// Mitsubishi GX Works2 project: Unloader Panel 23.07.21   PLC: Q03UDV
// Unloader Panel 23.07.21

PROGRAM MAIN
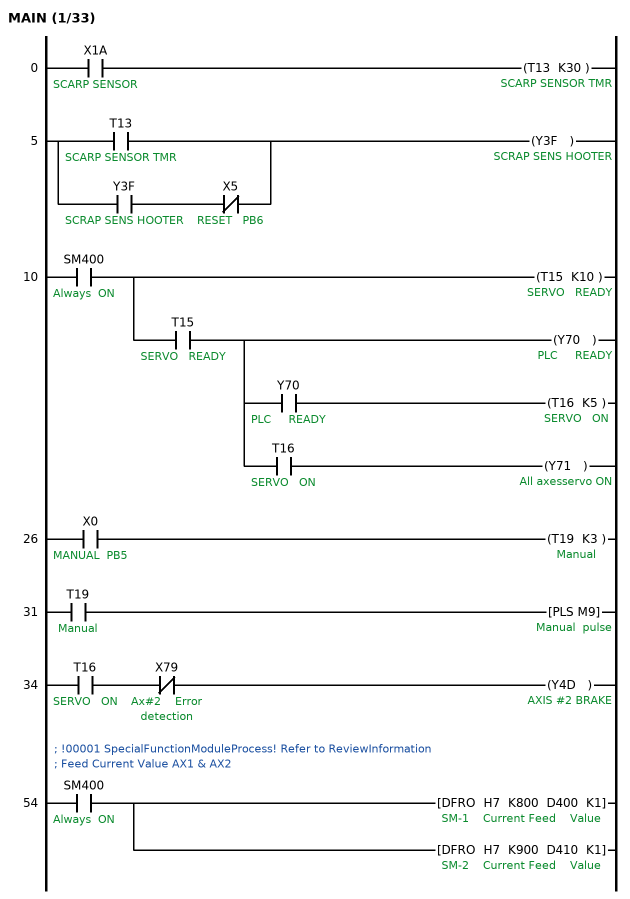
0     LD      X1A  ; SCARP SENSOR
      OUT     T13 K30  ; SCARP SENSOR TMR
5     LD      T13  ; SCARP SENSOR TMR
      LD      Y3F  ; SCRAP SENS HOOTER
      ANI     X5  ; RESET   PB6
      ORB
      OUT     Y3F  ; SCRAP SENS HOOTER
10    LD      SM400  ; Always  ON
      OUT     T15 K10  ; SERVO   READY
      AND     T15  ; SERVO   READY
      OUT     Y70  ; PLC     READY
      MPS
      AND     Y70  ; PLC     READY
      OUT     T16 K5  ; SERVO   ON
      MPP
      AND     T16  ; SERVO   ON
      OUT     Y71  ; All axesservo ON
26    LD      X0  ; MANUAL  PB5
      OUT     T19 K3  ; Manual
31    LD      T19  ; Manual
      PLS     M9  ; Manual  pulse
34    LD      T16  ; SERVO   ON
      ANI     X79  ; Ax#2    Error   detection
      OUT     Y4D  ; AXIS #2 BRAKE
; !00001 SpecialFunctionModuleProcess! Refer to ReviewInformation
; Feed Current Value AX1 & AX2
54    LD      SM400  ; Always  ON
      DFRO    H7 K800 D400 K1  ; SM-1    Current Feed    Value
      DFRO    H7 K900 D410 K1  ; SM-2    Current Feed    Value
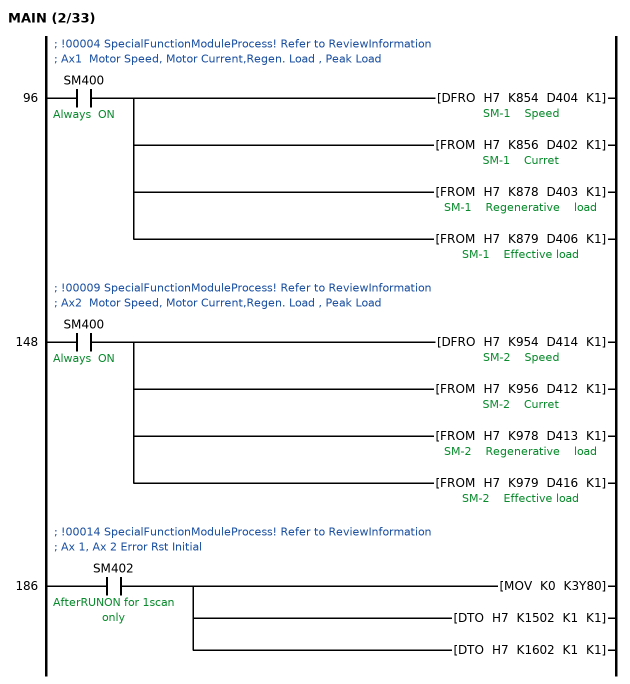
; !00004 SpecialFunctionModuleProcess! Refer to ReviewInformation
; Ax1  Motor Speed, Motor Current,Regen. Load , Peak Load
96    LD      SM400  ; Always  ON
      DFRO    H7 K854 D404 K1  ; SM-1    Speed
      FROM    H7 K856 D402 K1  ; SM-1    Curret
      FROM    H7 K878 D403 K1  ; SM-1    Regenerative    load
      FROM    H7 K879 D406 K1  ; SM-1    Effective load
; !00009 SpecialFunctionModuleProcess! Refer to ReviewInformation
; Ax2  Motor Speed, Motor Current,Regen. Load , Peak Load
148   LD      SM400  ; Always  ON
      DFRO    H7 K954 D414 K1  ; SM-2    Speed
      FROM    H7 K956 D412 K1  ; SM-2    Curret
      FROM    H7 K978 D413 K1  ; SM-2    Regenerative    load
      FROM    H7 K979 D416 K1  ; SM-2    Effective load
; !00014 SpecialFunctionModuleProcess! Refer to ReviewInformation
; Ax 1, Ax 2 Error Rst Initial
186   LD      SM402  ; AfterRUNON for 1scan    only
      MOV     K0 K3Y80  ; Axis #1 Positioning start
      DTO     H7 K1502 K1 K1
      DTO     H7 K1602 K1 K1
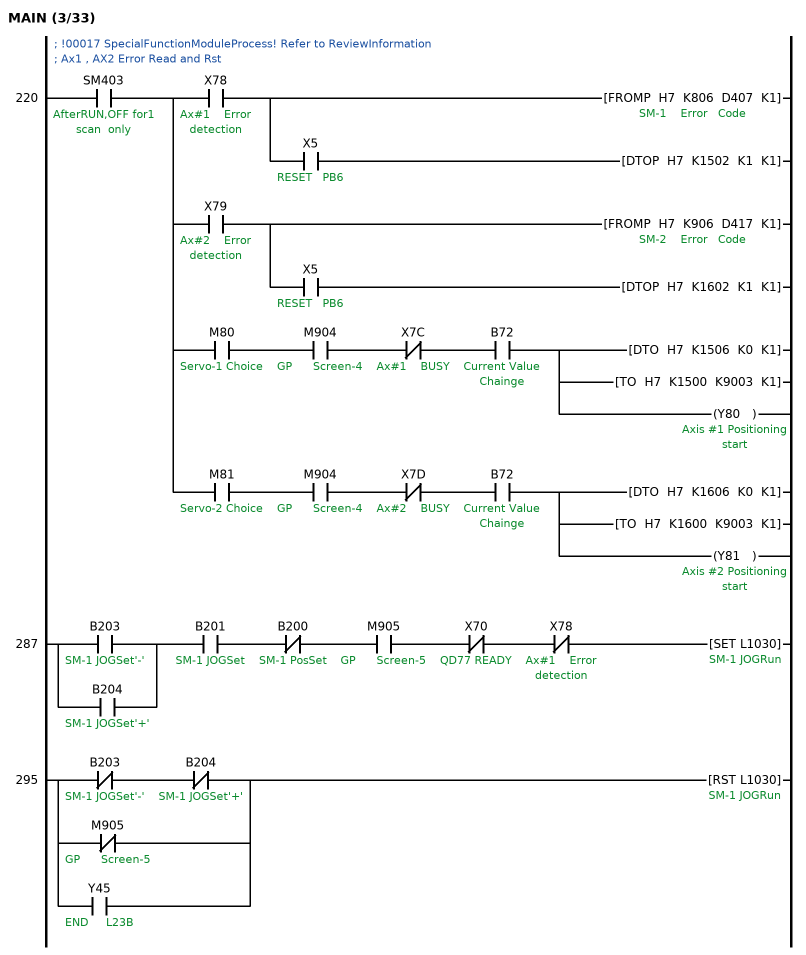
; !00017 SpecialFunctionModuleProcess! Refer to ReviewInformation
; Ax1 , AX2 Error Read and Rst
220   LD      SM403  ; AfterRUN,OFF for1 scan  only
      MPS
      AND     X78  ; Ax#1    Error   detection
      FROMP   H7 K806 D407 K1  ; SM-1    Error   Code
      AND     X5  ; RESET   PB6
      DTOP    H7 K1502 K1 K1
      MRD
      AND     X79  ; Ax#2    Error   detection
      FROMP   H7 K906 D417 K1  ; SM-2    Error   Code
      AND     X5  ; RESET   PB6
      DTOP    H7 K1602 K1 K1
      MRD
      AND     M80  ; Servo-1 Choice
      AND     M904  ; GP      Screen-4
      ANI     X7C  ; Ax#1    BUSY
      AND     B72  ; Current Value   Chainge
      DTO     H7 K1506 K0 K1
      TO      H7 K1500 K9003 K1
      OUT     Y80  ; Axis #1 Positioning start
      MPP
      AND     M81  ; Servo-2 Choice
      AND     M904  ; GP      Screen-4
      ANI     X7D  ; Ax#2    BUSY
      AND     B72  ; Current Value   Chainge
      DTO     H7 K1606 K0 K1
      TO      H7 K1600 K9003 K1
      OUT     Y81  ; Axis #2 Positioning start
287   LD      B203  ; SM-1 JOGSet'-'
      OR      B204  ; SM-1 JOGSet'+'
      AND     B201  ; SM-1 JOGSet
      ANI     B200  ; SM-1 PosSet
      AND     M905  ; GP      Screen-5
      ANI     X70  ; QD77 READY
      ANI     X78  ; Ax#1    Error   detection
      SET     L1030  ; SM-1 JOGRun
295   LDI     B203  ; SM-1 JOGSet'-'
      ANI     B204  ; SM-1 JOGSet'+'
      ORI     M905  ; GP      Screen-5
      OR      Y45  ; END     L23B
      RST     L1030  ; SM-1 JOGRun
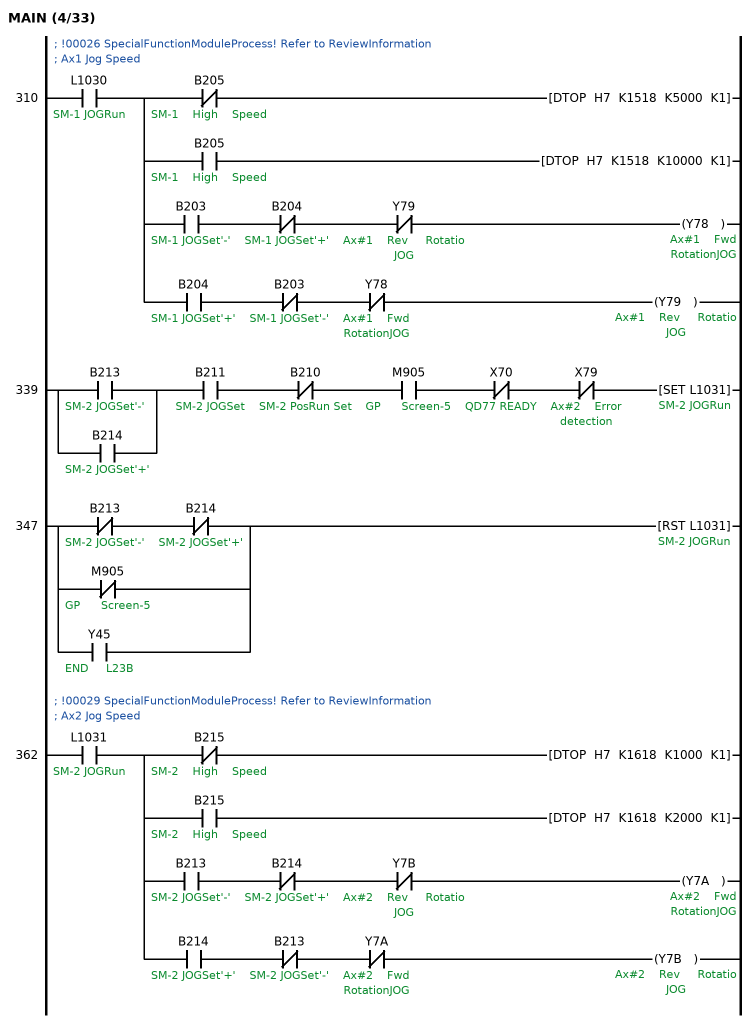
; !00026 SpecialFunctionModuleProcess! Refer to ReviewInformation
; Ax1 Jog Speed
310   LD      L1030  ; SM-1 JOGRun
      MPS
      ANI     B205  ; SM-1    High    Speed
      DTOP    H7 K1518 K5000 K1
      MRD
      AND     B205  ; SM-1    High    Speed
      DTOP    H7 K1518 K10000 K1
      MRD
      AND     B203  ; SM-1 JOGSet'-'
      ANI     B204  ; SM-1 JOGSet'+'
      ANI     Y79  ; Ax#1    Rev     Rotatio JOG
      OUT     Y78  ; Ax#1    Fwd     RotationJOG
      MPP
      AND     B204  ; SM-1 JOGSet'+'
      ANI     B203  ; SM-1 JOGSet'-'
      ANI     Y78  ; Ax#1    Fwd     RotationJOG
      OUT     Y79  ; Ax#1    Rev     Rotatio JOG
339   LD      B213  ; SM-2 JOGSet'-'
      OR      B214  ; SM-2 JOGSet'+'
      AND     B211  ; SM-2 JOGSet
      ANI     B210  ; SM-2 PosRun Set
      AND     M905  ; GP      Screen-5
      ANI     X70  ; QD77 READY
      ANI     X79  ; Ax#2    Error   detection
      SET     L1031  ; SM-2 JOGRun
347   LDI     B213  ; SM-2 JOGSet'-'
      ANI     B214  ; SM-2 JOGSet'+'
      ORI     M905  ; GP      Screen-5
      OR      Y45  ; END     L23B
      RST     L1031  ; SM-2 JOGRun
; !00029 SpecialFunctionModuleProcess! Refer to ReviewInformation
; Ax2 Jog Speed
362   LD      L1031  ; SM-2 JOGRun
      MPS
      ANI     B215  ; SM-2    High    Speed
      DTOP    H7 K1618 K1000 K1
      MRD
      AND     B215  ; SM-2    High    Speed
      DTOP    H7 K1618 K2000 K1
      MRD
      AND     B213  ; SM-2 JOGSet'-'
      ANI     B214  ; SM-2 JOGSet'+'
      ANI     Y7B  ; Ax#2    Rev     Rotatio JOG
      OUT     Y7A  ; Ax#2    Fwd     RotationJOG
      MPP
      AND     B214  ; SM-2 JOGSet'+'
      ANI     B213  ; SM-2 JOGSet'-'
      ANI     Y7A  ; Ax#2    Fwd     RotationJOG
      OUT     Y7B  ; Ax#2    Rev     Rotatio JOG
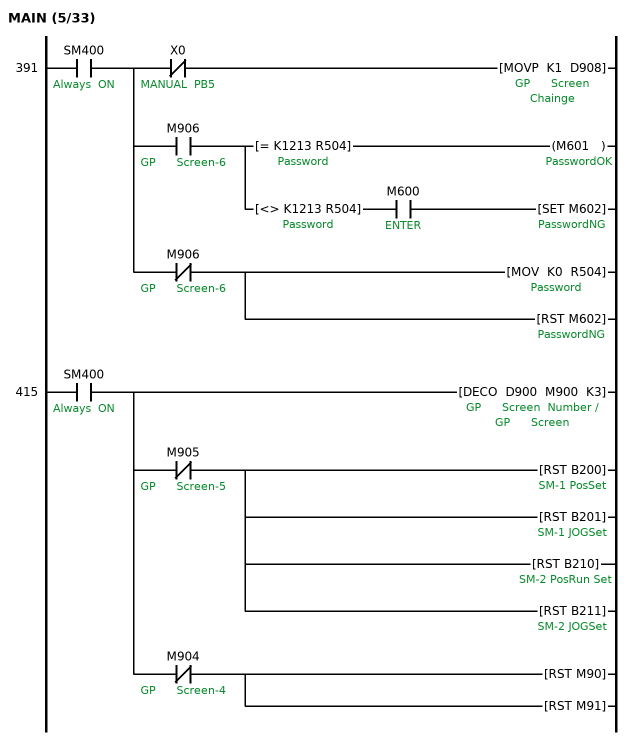
391   LD      SM400  ; Always  ON
      MPS
      ANI     X0  ; MANUAL  PB5
      MOVP    K1 D908  ; GP      Screen  Chainge
      MRD
      AND     M906  ; GP      Screen-6
      MPS
      AND=    K1213 R504  ; Password
      OUT     M601  ; PasswordOK
      MPP
      AND<>   K1213 R504  ; Password
      AND     M600  ; ENTER
      SET     M602  ; PasswordNG
      MPP
      ANI     M906  ; GP      Screen-6
      MOV     K0 R504
      RST     M602  ; PasswordNG
415   LD      SM400  ; Always  ON
      DECO    D900 M900 K3  ; GP      Screen  Number / GP      Screen
      MPS
      ANI     M905  ; GP      Screen-5
      RST     B200  ; SM-1 PosSet
      RST     B201  ; SM-1 JOGSet
      RST     B210  ; SM-2 PosRun Set
      RST     B211  ; SM-2 JOGSet
      MPP
      ANI     M904  ; GP      Screen-4
      RST     M90
      RST     M91
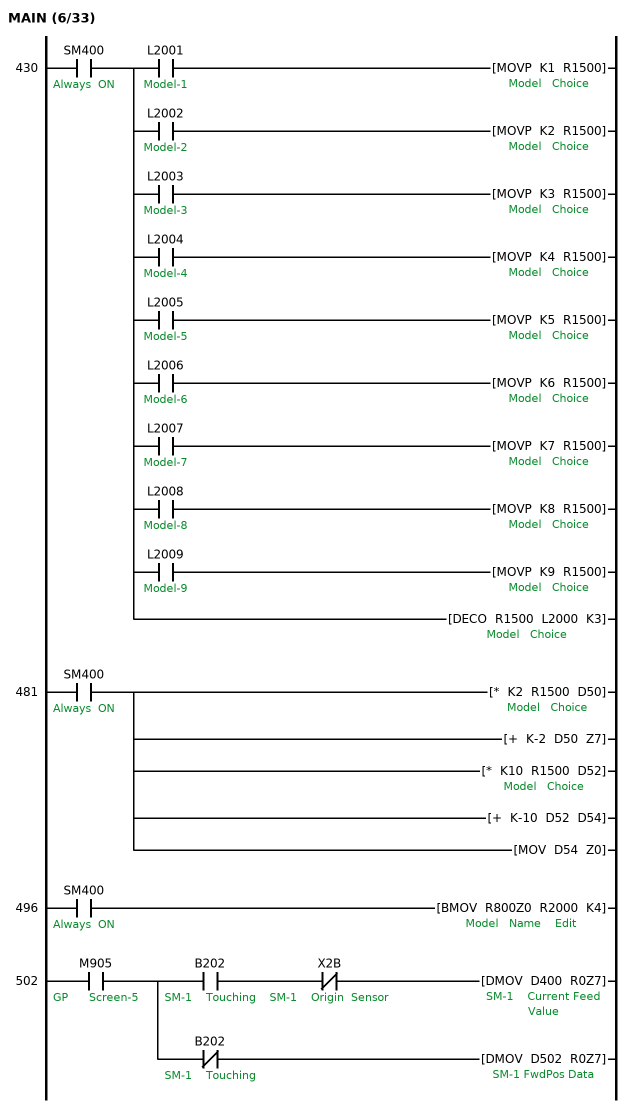
430   LD      SM400  ; Always  ON
      MPS
      AND     L2001  ; Model-1
      MOVP    K1 R1500  ; Model   Choice
      MRD
      AND     L2002  ; Model-2
      MOVP    K2 R1500
      MRD
      AND     L2003  ; Model-3
      MOVP    K3 R1500
      MRD
      AND     L2004  ; Model-4
      MOVP    K4 R1500
      MRD
      AND     L2005  ; Model-5
      MOVP    K5 R1500
      MRD
      AND     L2006  ; Model-6
      MOVP    K6 R1500
      MRD
      AND     L2007  ; Model-7
      MOVP    K7 R1500
      MRD
      AND     L2008  ; Model-8
      MOVP    K8 R1500
      MRD
      AND     L2009  ; Model-9
      MOVP    K9 R1500
      MPP
      DECO    R1500 L2000 K3
481   LD      SM400  ; Always  ON
      *       K2 R1500 D50
      +       K-2 D50 Z7
      *       K10 R1500 D52
      +       K-10 D52 D54
      MOV     D54 Z0
496   LD      SM400  ; Always  ON
      BMOV    R800Z0 R2000 K4  ; Model   Name    Edit
502   LD      M905  ; GP      Screen-5
      MPS
      AND     B202  ; SM-1    Touching
      ANI     X2B  ; SM-1    Origin  Sensor
      DMOV    D400 R0Z7
      MPP
      ANI     B202  ; SM-1    Touching
      DMOV    D502 R0Z7  ; SM-1 FwdPos Data
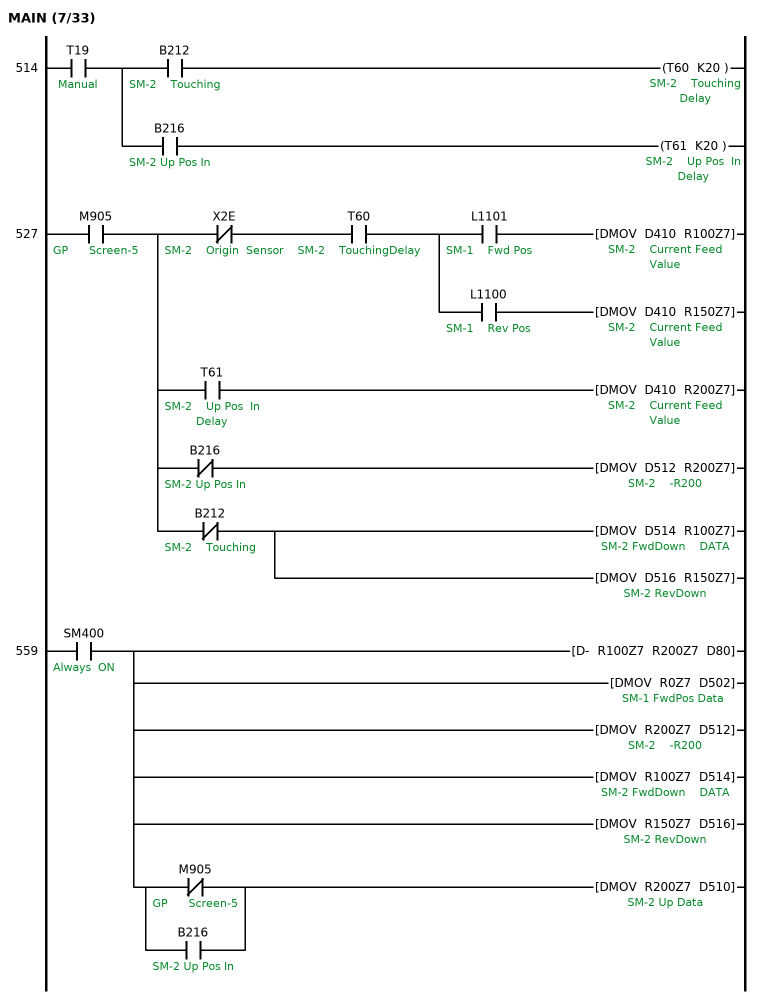
514   LD      T19  ; Manual
      MPS
      AND     B212  ; SM-2    Touching
      OUT     T60 K20  ; SM-2    TouchingDelay
      MPP
      AND     B216  ; SM-2 Up Pos In
      OUT     T61 K20  ; SM-2    Up Pos  In Delay
527   LD      M905  ; GP      Screen-5
      MPS
      ANI     X2E  ; SM-2    Origin  Sensor
      AND     T60  ; SM-2    TouchingDelay
      MPS
      AND     L1101  ; SM-1    Fwd Pos
      DMOV    D410 R100Z7
      MPP
      AND     L1100  ; SM-1    Rev Pos
      DMOV    D410 R150Z7
      MRD
      AND     T61  ; SM-2    Up Pos  In Delay
      DMOV    D410 R200Z7
      MRD
      ANI     B216  ; SM-2 Up Pos In
      DMOV    D512 R200Z7  ; SM-2    -R200
      MPP
      ANI     B212  ; SM-2    Touching
      DMOV    D514 R100Z7  ; SM-2 FwdDown    DATA
      DMOV    D516 R150Z7  ; SM-2 RevDown
559   LD      SM400  ; Always  ON
      D-      R100Z7 R200Z7 D80
      DMOV    R0Z7 D502
      DMOV    R200Z7 D512
      DMOV    R100Z7 D514
      DMOV    R150Z7 D516
      LDI     M905  ; GP      Screen-5
      OR      B216  ; SM-2 Up Pos In
      ANB
      DMOV    R200Z7 D510  ; SM-2 Up Data
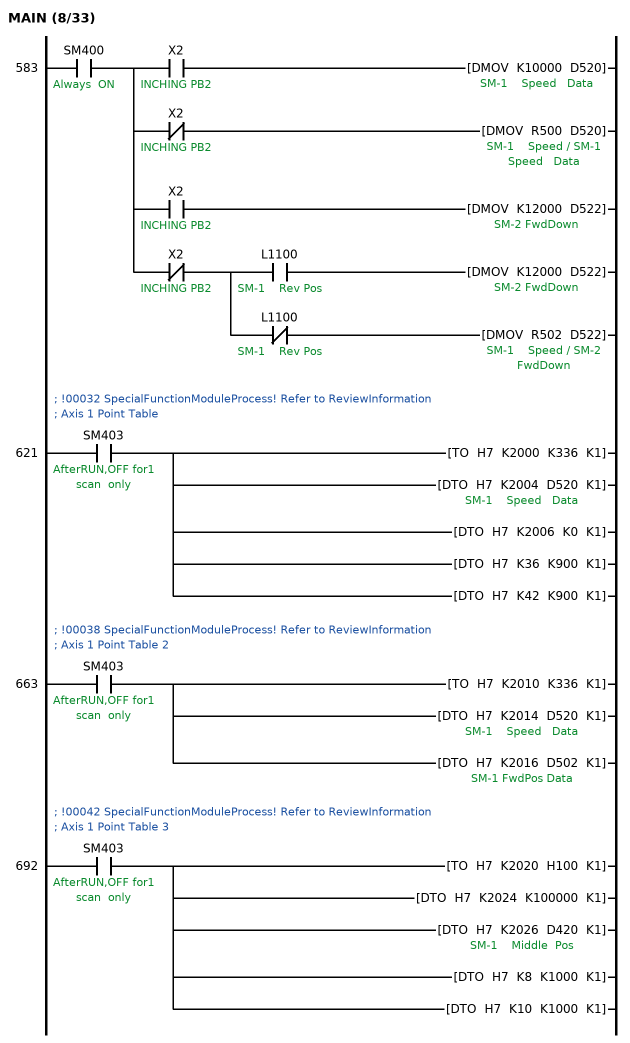
583   LD      SM400  ; Always  ON
      MPS
      AND     X2  ; INCHING PB2
      DMOV    K10000 D520  ; SM-1    Speed   Data
      MRD
      ANI     X2  ; INCHING PB2
      DMOV    R500 D520  ; SM-1    Speed
      MRD
      AND     X2  ; INCHING PB2
      DMOV    K12000 D522  ; SM-2 FwdDown
      MPP
      ANI     X2  ; INCHING PB2
      MPS
      AND     L1100  ; SM-1    Rev Pos
      DMOV    K12000 D522
      MPP
      ANI     L1100  ; SM-1    Rev Pos
      DMOV    R502 D522  ; SM-1    Speed
; !00032 SpecialFunctionModuleProcess! Refer to ReviewInformation
; Axis 1 Point Table
621   LD      SM403  ; AfterRUN,OFF for1 scan  only
      TO      H7 K2000 K336 K1
      DTO     H7 K2004 D520 K1
      DTO     H7 K2006 K0 K1
      DTO     H7 K36 K900 K1
      DTO     H7 K42 K900 K1
; !00038 SpecialFunctionModuleProcess! Refer to ReviewInformation
; Axis 1 Point Table 2
663   LD      SM403  ; AfterRUN,OFF for1 scan  only
      TO      H7 K2010 K336 K1
      DTO     H7 K2014 D520 K1
      DTO     H7 K2016 D502 K1
; !00042 SpecialFunctionModuleProcess! Refer to ReviewInformation
; Axis 1 Point Table 3
692   LD      SM403  ; AfterRUN,OFF for1 scan  only
      TO      H7 K2020 H100 K1
      DTO     H7 K2024 K100000 K1
      DTO     H7 K2026 D420 K1  ; SM-1    Middle  Pos
      DTO     H7 K8 K1000 K1
      DTO     H7 K10 K1000 K1
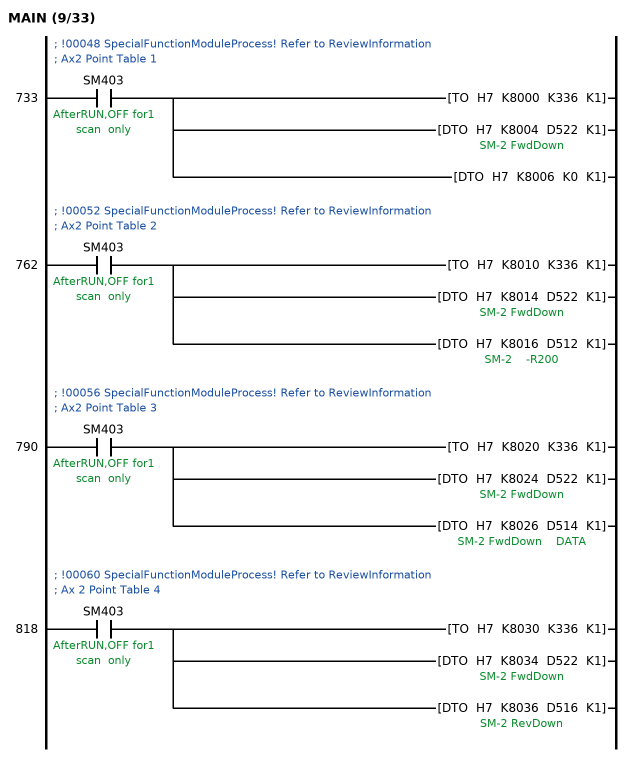
; !00048 SpecialFunctionModuleProcess! Refer to ReviewInformation
; Ax2 Point Table 1
733   LD      SM403  ; AfterRUN,OFF for1 scan  only
      TO      H7 K8000 K336 K1
      DTO     H7 K8004 D522 K1
      DTO     H7 K8006 K0 K1
; !00052 SpecialFunctionModuleProcess! Refer to ReviewInformation
; Ax2 Point Table 2
762   LD      SM403  ; AfterRUN,OFF for1 scan  only
      TO      H7 K8010 K336 K1
      DTO     H7 K8014 D522 K1
      DTO     H7 K8016 D512 K1
; !00056 SpecialFunctionModuleProcess! Refer to ReviewInformation
; Ax2 Point Table 3
790   LD      SM403  ; AfterRUN,OFF for1 scan  only
      TO      H7 K8020 K336 K1
      DTO     H7 K8024 D522 K1
      DTO     H7 K8026 D514 K1
; !00060 SpecialFunctionModuleProcess! Refer to ReviewInformation
; Ax 2 Point Table 4
818   LD      SM403  ; AfterRUN,OFF for1 scan  only
      TO      H7 K8030 K336 K1
      DTO     H7 K8034 D522 K1
      DTO     H7 K8036 D516 K1
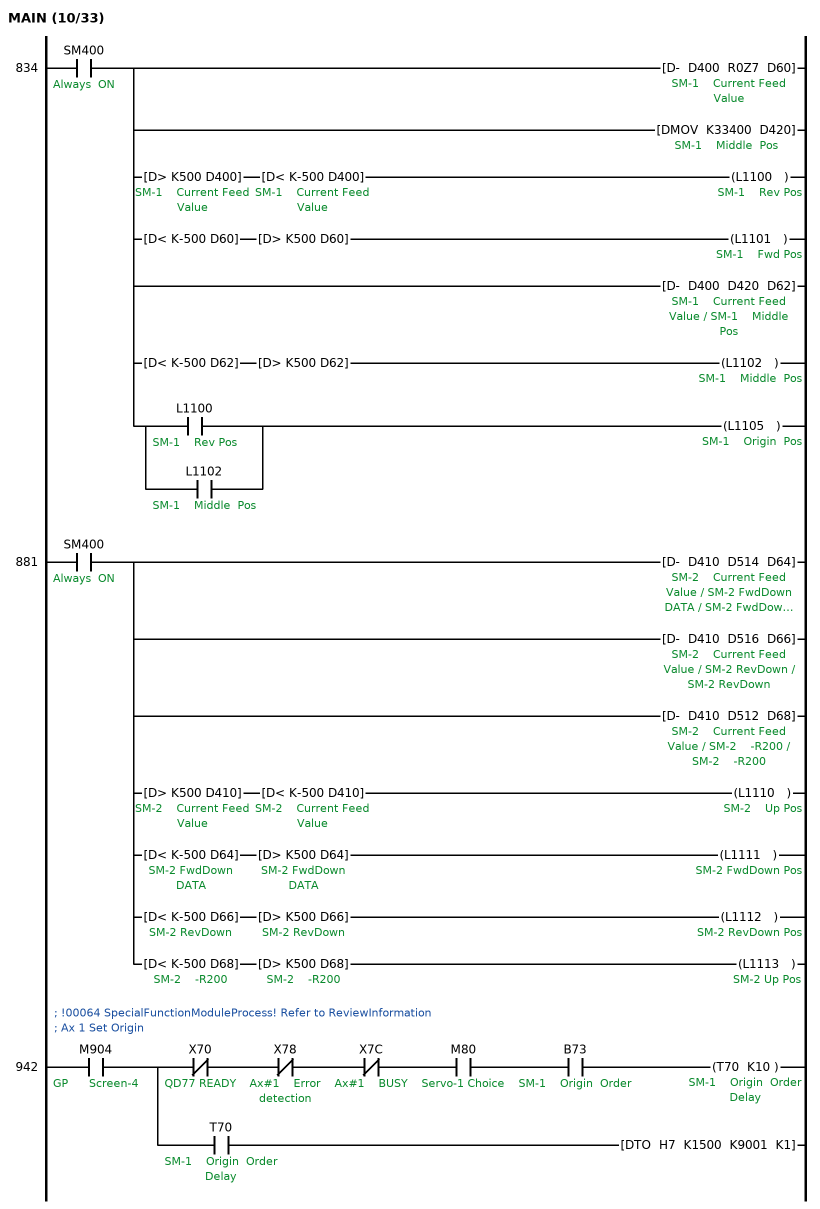
834   LD      SM400  ; Always  ON
      D-      D400 R0Z7 D60
      DMOV    K33400 D420
      MPS
      ANDD>   K500 D400  ; SM-1    Current Feed    Value
      ANDD<   K-500 D400  ; SM-1    Current Feed    Value
      OUT     L1100  ; SM-1    Rev Pos
      MRD
      ANDD<   K-500 D60
      ANDD>   K500 D60
      OUT     L1101  ; SM-1    Fwd Pos
      MPP
      D-      D400 D420 D62
      MPS
      ANDD<   K-500 D62
      ANDD>   K500 D62
      OUT     L1102  ; SM-1    Middle  Pos
      MPP
      LD      L1100  ; SM-1    Rev Pos
      OR      L1102  ; SM-1    Middle  Pos
      ANB
      OUT     L1105  ; SM-1    Origin  Pos
881   LD      SM400  ; Always  ON
      D-      D410 D514 D64  ; SM-2 FwdDown    DATA
      D-      D410 D516 D66  ; SM-2 RevDown
      D-      D410 D512 D68  ; SM-2    -R200
      MPS
      ANDD>   K500 D410  ; SM-2    Current Feed    Value
      ANDD<   K-500 D410  ; SM-2    Current Feed    Value
      OUT     L1110  ; SM-2    Up Pos
      MRD
      ANDD<   K-500 D64  ; SM-2 FwdDown    DATA
      ANDD>   K500 D64  ; SM-2 FwdDown    DATA
      OUT     L1111  ; SM-2 FwdDown Pos
      MRD
      ANDD<   K-500 D66  ; SM-2 RevDown
      ANDD>   K500 D66  ; SM-2 RevDown
      OUT     L1112  ; SM-2 RevDown Pos
      MPP
      ANDD<   K-500 D68  ; SM-2    -R200
      ANDD>   K500 D68  ; SM-2    -R200
      OUT     L1113  ; SM-2 Up Pos
; !00064 SpecialFunctionModuleProcess! Refer to ReviewInformation
; Ax 1 Set Origin
942   LD      M904  ; GP      Screen-4
      MPS
      ANI     X70  ; QD77 READY
      ANI     X78  ; Ax#1    Error   detection
      ANI     X7C  ; Ax#1    BUSY
      AND     M80  ; Servo-1 Choice
      AND     B73  ; SM-1    Origin  Order
      OUT     T70 K10  ; SM-1    Origin  Order   Delay
      MPP
      AND     T70  ; SM-1    Origin  Order   Delay
      DTO     H7 K1500 K9001 K1
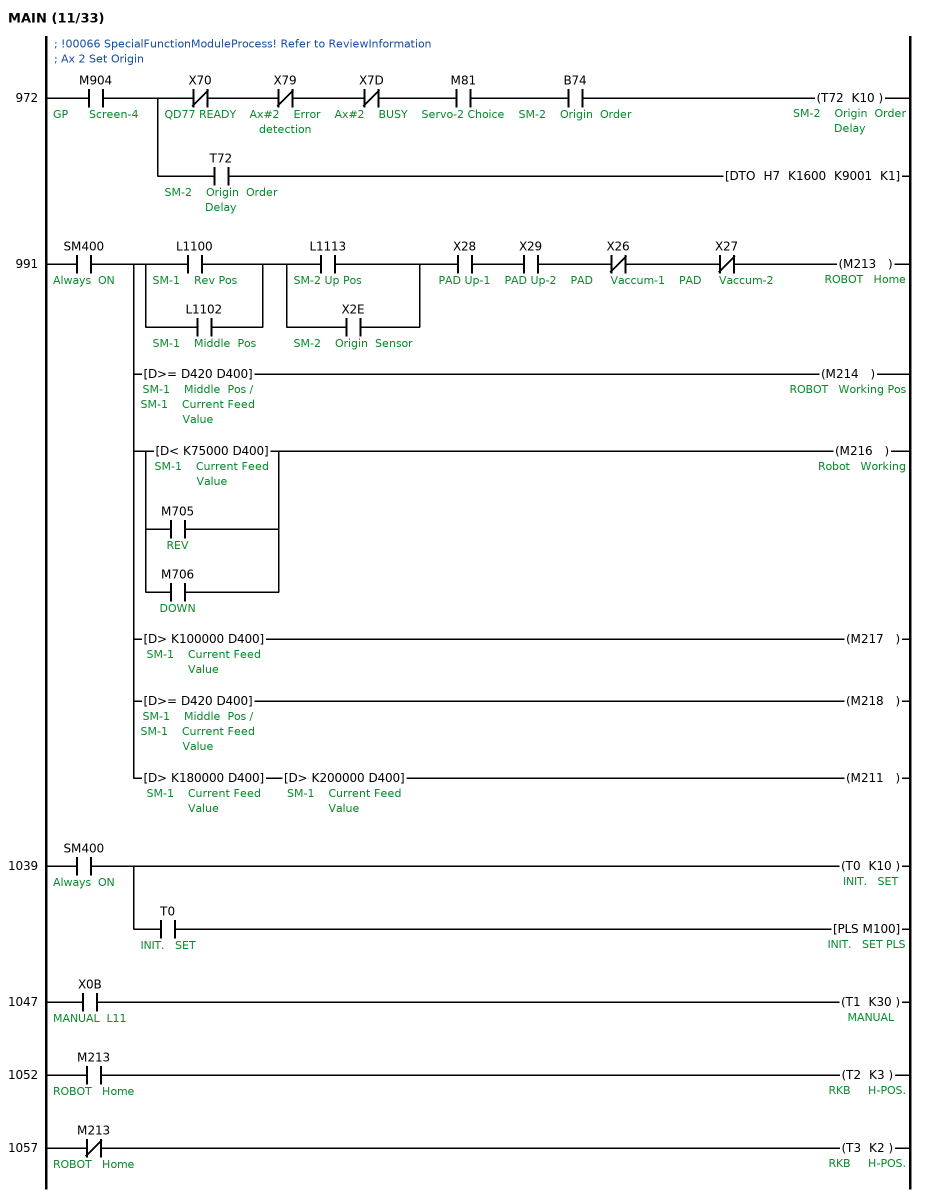
; !00066 SpecialFunctionModuleProcess! Refer to ReviewInformation
; Ax 2 Set Origin
972   LD      M904  ; GP      Screen-4
      MPS
      ANI     X70  ; QD77 READY
      ANI     X79  ; Ax#2    Error   detection
      ANI     X7D  ; Ax#2    BUSY
      AND     M81  ; Servo-2 Choice
      AND     B74  ; SM-2    Origin  Order
      OUT     T72 K10  ; SM-2    Origin  Order   Delay
      MPP
      AND     T72  ; SM-2    Origin  Order   Delay
      DTO     H7 K1600 K9001 K1
991   LD      SM400  ; Always  ON
      MPS
      LD      L1100  ; SM-1    Rev Pos
      OR      L1102  ; SM-1    Middle  Pos
      ANB
      LD      L1113  ; SM-2 Up Pos
      OR      X2E  ; SM-2    Origin  Sensor
      ANB
      AND     X28  ; PAD Up-1
      AND     X29  ; PAD Up-2
      ANI     X26  ; PAD     Vaccum-1
      ANI     X27  ; PAD     Vaccum-2
      OUT     M213  ; ROBOT   Home
      MRD
      ANDD>=  D420 D400  ; SM-1    Middle  Pos / SM-1    Current Feed    Value
      OUT     M214  ; ROBOT   Working Pos
      MRD
      LDD<    K75000 D400  ; SM-1    Current Feed    Value
      OR      M705  ; REV
      OR      M706  ; DOWN
      ANB
      OUT     M216  ; Robot   Working
      MRD
      ANDD>   K100000 D400  ; SM-1    Current Feed    Value
      OUT     M217
      MRD
      ANDD>=  D420 D400  ; SM-1    Middle  Pos / SM-1    Current Feed    Value
      OUT     M218
      MPP
      ANDD>   K180000 D400  ; SM-1    Current Feed    Value
      ANDD>   K200000 D400  ; SM-1    Current Feed    Value
      OUT     M211
1039  LD      SM400  ; Always  ON
      OUT     T0 K10  ; INIT.   SET
      AND     T0  ; INIT.   SET
      PLS     M100  ; INIT.   SET PLS
1047  LD      X0B  ; MANUAL  L11
      OUT     T1 K30  ; MANUAL
1052  LD      M213  ; ROBOT   Home
      OUT     T2 K3  ; RKB     H-POS.
1057  LDI     M213  ; ROBOT   Home
      OUT     T3 K2  ; RKB     H-POS.
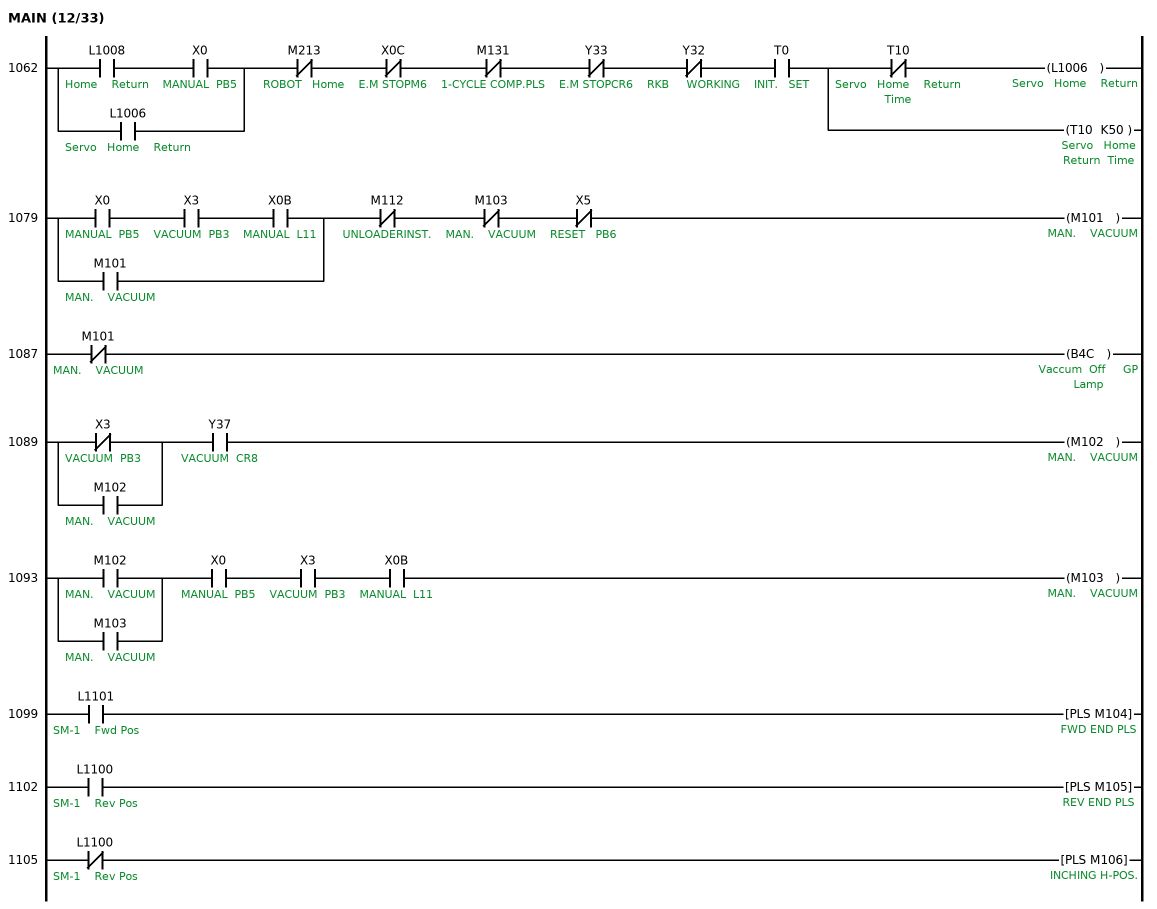
1062  LD      L1008  ; Home    Return
      AND     X0  ; MANUAL  PB5
      OR      L1006  ; Servo   Home    Return
      ANI     M213  ; ROBOT   Home
      ANI     X0C  ; E.M STOPM6
      ANI     M131  ; 1-CYCLE COMP.PLS
      ANI     Y33  ; E.M STOPCR6
      ANI     Y32  ; RKB     WORKING
      AND     T0  ; INIT.   SET
      MPS
      ANI     T10  ; Servo   Home    Return  Time
      OUT     L1006  ; Servo   Home    Return
      MPP
      OUT     T10 K50  ; Servo   Home    Return  Time
1079  LD      X0  ; MANUAL  PB5
      AND     X3  ; VACUUM  PB3
      AND     X0B  ; MANUAL  L11
      OR      M101  ; MAN.    VACUUM
      ANI     M112  ; UNLOADERINST.
      ANI     M103  ; MAN.    VACUUM
      ANI     X5  ; RESET   PB6
      OUT     M101  ; MAN.    VACUUM
1087  LDI     M101  ; MAN.    VACUUM
      OUT     B4C  ; Vaccum  Off     GP Lamp
1089  LDI     X3  ; VACUUM  PB3
      OR      M102  ; MAN.    VACUUM
      AND     Y37  ; VACUUM  CR8
      OUT     M102  ; MAN.    VACUUM
1093  LD      M102  ; MAN.    VACUUM
      OR      M103  ; MAN.    VACUUM
      AND     X0  ; MANUAL  PB5
      AND     X3  ; VACUUM  PB3
      AND     X0B  ; MANUAL  L11
      OUT     M103  ; MAN.    VACUUM
1099  LD      L1101  ; SM-1    Fwd Pos
      PLS     M104  ; FWD END PLS
1102  LD      L1100  ; SM-1    Rev Pos
      PLS     M105  ; REV END PLS
1105  LDI     L1100  ; SM-1    Rev Pos
      PLS     M106  ; INCHING H-POS.
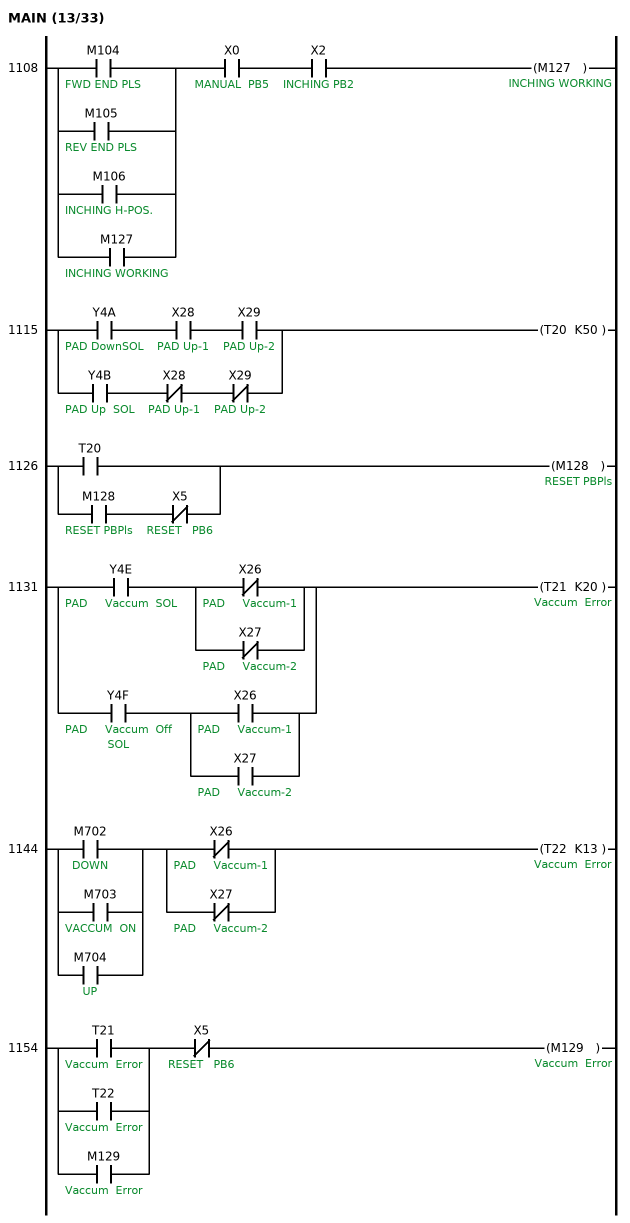
1108  LD      M104  ; FWD END PLS
      OR      M105  ; REV END PLS
      OR      M106  ; INCHING H-POS.
      OR      M127  ; INCHING WORKING
      AND     X0  ; MANUAL  PB5
      AND     X2  ; INCHING PB2
      OUT     M127  ; INCHING WORKING
1115  LD      Y4A  ; PAD DownSOL
      AND     X28  ; PAD Up-1
      AND     X29  ; PAD Up-2
      LD      Y4B  ; PAD Up  SOL
      ANI     X28  ; PAD Up-1
      ANI     X29  ; PAD Up-2
      ORB
      OUT     T20 K50
1126  LD      T20
      LD      M128  ; RESET PBPls
      ANI     X5  ; RESET   PB6
      ORB
      OUT     M128  ; RESET PBPls
1131  LD      Y4E  ; PAD     Vaccum  SOL
      LDI     X26  ; PAD     Vaccum-1
      ORI     X27  ; PAD     Vaccum-2
      ANB
      LD      Y4F  ; PAD     Vaccum  Off SOL
      LD      X26  ; PAD     Vaccum-1
      OR      X27  ; PAD     Vaccum-2
      ANB
      ORB
      OUT     T21 K20  ; Vaccum  Error
1144  LD      M702  ; DOWN
      OR      M703  ; VACCUM  ON
      OR      M704  ; UP
      LDI     X26  ; PAD     Vaccum-1
      ORI     X27  ; PAD     Vaccum-2
      ANB
      OUT     T22 K13  ; Vaccum  Error
1154  LD      T21  ; Vaccum  Error
      OR      T22  ; Vaccum  Error
      OR      M129  ; Vaccum  Error
      ANI     X5  ; RESET   PB6
      OUT     M129  ; Vaccum  Error
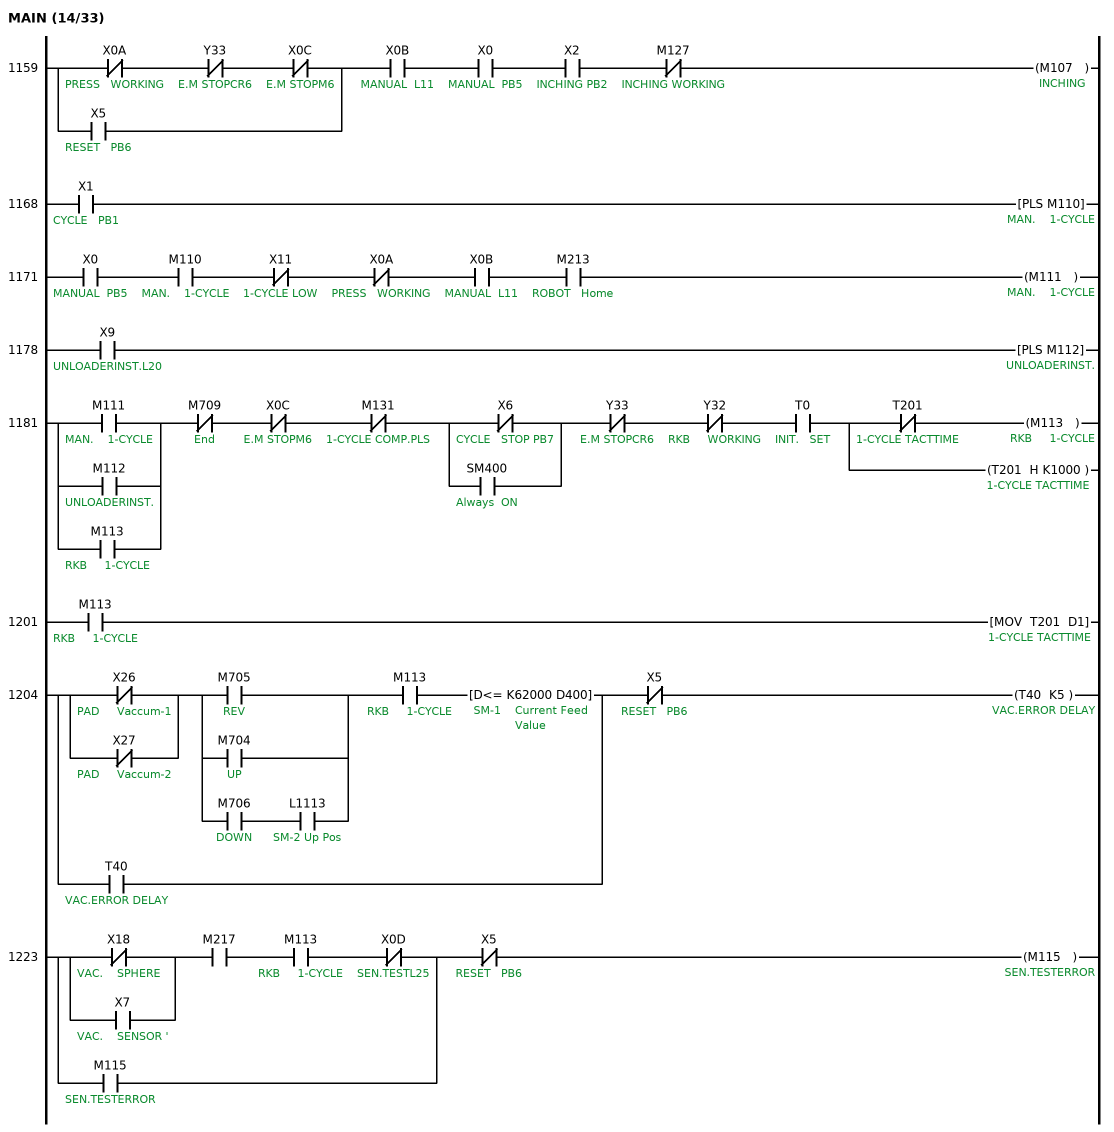
1159  LDI     X0A  ; PRESS   WORKING
      ANI     Y33  ; E.M STOPCR6
      ANI     X0C  ; E.M STOPM6
      OR      X5  ; RESET   PB6
      AND     X0B  ; MANUAL  L11
      AND     X0  ; MANUAL  PB5
      AND     X2  ; INCHING PB2
      ANI     M127  ; INCHING WORKING
      OUT     M107  ; INCHING
1168  LD      X1  ; CYCLE   PB1
      PLS     M110  ; MAN.    1-CYCLE
1171  LD      X0  ; MANUAL  PB5
      AND     M110  ; MAN.    1-CYCLE
      ANI     X11  ; 1-CYCLE LOW
      ANI     X0A  ; PRESS   WORKING
      AND     X0B  ; MANUAL  L11
      AND     M213  ; ROBOT   Home
      OUT     M111  ; MAN.    1-CYCLE
1178  LD      X9  ; UNLOADERINST.L20
      PLS     M112  ; UNLOADERINST.
1181  LD      M111  ; MAN.    1-CYCLE
      OR      M112  ; UNLOADERINST.
      OR      M113  ; RKB     1-CYCLE
      ANI     M709  ; End
      ANI     X0C  ; E.M STOPM6
      ANI     M131  ; 1-CYCLE COMP.PLS
      LDI     X6  ; CYCLE   STOP PB7
      OR      SM400  ; Always  ON
      ANB
      ANI     Y33  ; E.M STOPCR6
      ANI     Y32  ; RKB     WORKING
      AND     T0  ; INIT.   SET
      MPS
      ANI     T201  ; 1-CYCLE TACTTIME
      OUT     M113  ; RKB     1-CYCLE
      MPP
      OUTH    T201 K1000  ; 1-CYCLE TACTTIME
1201  LD      M113  ; RKB     1-CYCLE
      MOV     T201 D1
1204  LDI     X26  ; PAD     Vaccum-1
      ORI     X27  ; PAD     Vaccum-2
      LD      M705  ; REV
      OR      M704  ; UP
      LD      M706  ; DOWN
      AND     L1113  ; SM-2 Up Pos
      ORB
      ANB
      AND     M113  ; RKB     1-CYCLE
      ANDD<=  K62000 D400  ; SM-1    Current Feed    Value
      OR      T40  ; VAC.ERROR DELAY
      ANI     X5  ; RESET   PB6
      OUT     T40 K5  ; VAC.ERROR DELAY
1223  LDI     X18  ; VAC.    SPHERE
      OR      X7  ; VAC.    SENSOR '
      AND     M217
      AND     M113  ; RKB     1-CYCLE
      ANI     X0D  ; SEN.TESTL25
      OR      M115  ; SEN.TESTERROR
      ANI     X5  ; RESET   PB6
      OUT     M115  ; SEN.TESTERROR
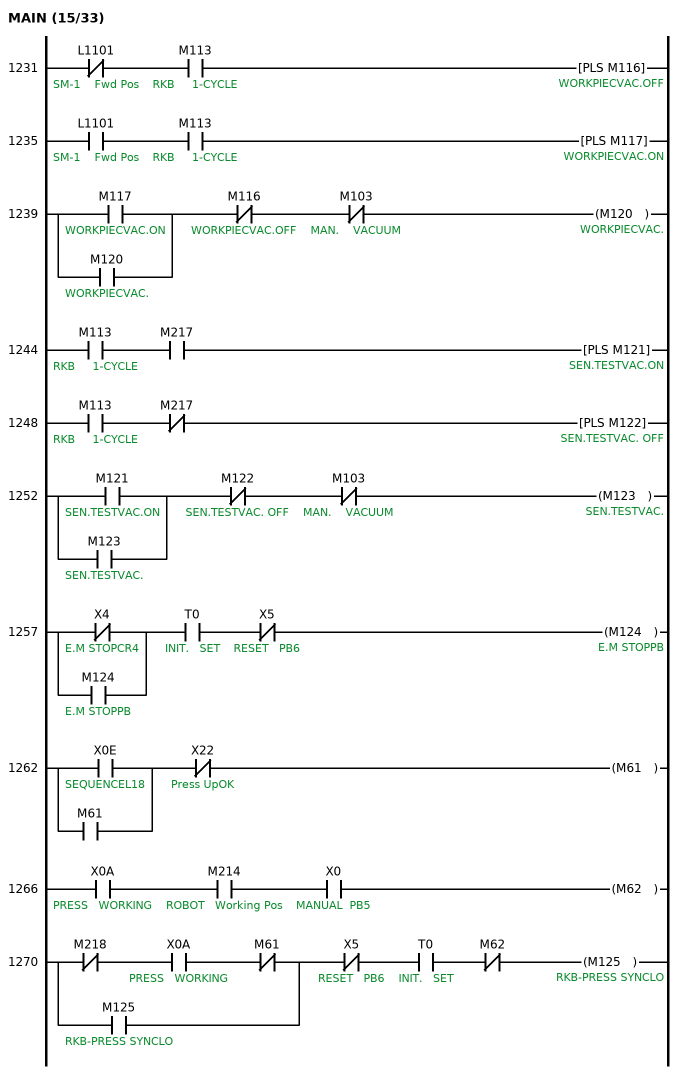
1231  LDI     L1101  ; SM-1    Fwd Pos
      AND     M113  ; RKB     1-CYCLE
      PLS     M116  ; WORKPIECVAC.OFF
1235  LD      L1101  ; SM-1    Fwd Pos
      AND     M113  ; RKB     1-CYCLE
      PLS     M117  ; WORKPIECVAC.ON
1239  LD      M117  ; WORKPIECVAC.ON
      OR      M120  ; WORKPIECVAC.
      ANI     M116  ; WORKPIECVAC.OFF
      ANI     M103  ; MAN.    VACUUM
      OUT     M120  ; WORKPIECVAC.
1244  LD      M113  ; RKB     1-CYCLE
      AND     M217
      PLS     M121  ; SEN.TESTVAC.ON
1248  LD      M113  ; RKB     1-CYCLE
      ANI     M217
      PLS     M122  ; SEN.TESTVAC. OFF
1252  LD      M121  ; SEN.TESTVAC.ON
      OR      M123  ; SEN.TESTVAC.
      ANI     M122  ; SEN.TESTVAC. OFF
      ANI     M103  ; MAN.    VACUUM
      OUT     M123  ; SEN.TESTVAC.
1257  LDI     X4  ; E.M STOPCR4
      OR      M124  ; E.M STOPPB
      AND     T0  ; INIT.   SET
      ANI     X5  ; RESET   PB6
      OUT     M124  ; E.M STOPPB
1262  LD      X0E  ; SEQUENCEL18
      OR      M61
      ANI     X22  ; Press UpOK
      OUT     M61
1266  LD      X0A  ; PRESS   WORKING
      AND     M214  ; ROBOT   Working Pos
      AND     X0  ; MANUAL  PB5
      OUT     M62
1270  LDI     M218
      AND     X0A  ; PRESS   WORKING
      ANI     M61
      OR      M125  ; RKB-PRESS SYNCLO
      ANI     X5  ; RESET   PB6
      AND     T0  ; INIT.   SET
      ANI     M62
      OUT     M125  ; RKB-PRESS SYNCLO
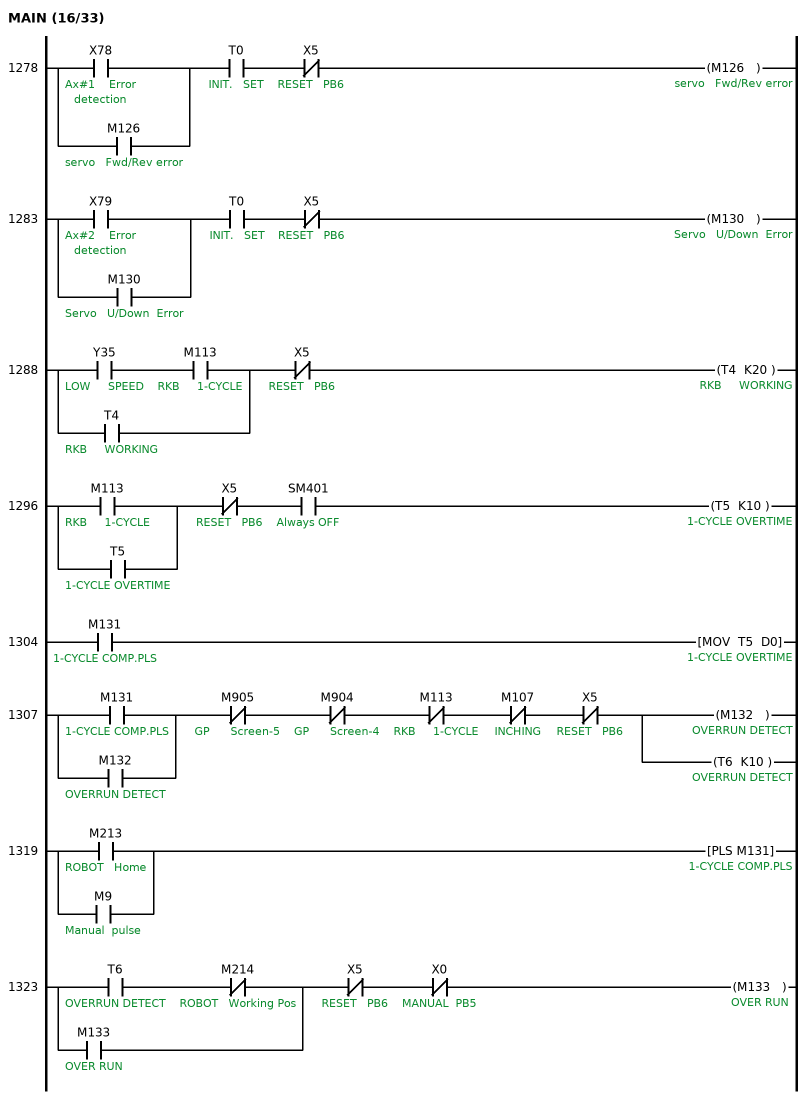
1278  LD      X78  ; Ax#1    Error   detection
      OR      M126  ; servo   Fwd/Rev error
      AND     T0  ; INIT.   SET
      ANI     X5  ; RESET   PB6
      OUT     M126  ; servo   Fwd/Rev error
1283  LD      X79  ; Ax#2    Error   detection
      OR      M130  ; Servo   U/Down  Error
      AND     T0  ; INIT.   SET
      ANI     X5  ; RESET   PB6
      OUT     M130  ; Servo   U/Down  Error
1288  LD      Y35  ; LOW     SPEED
      AND     M113  ; RKB     1-CYCLE
      OR      T4  ; RKB     WORKING
      ANI     X5  ; RESET   PB6
      OUT     T4 K20  ; RKB     WORKING
1296  LD      M113  ; RKB     1-CYCLE
      OR      T5  ; 1-CYCLE OVERTIME
      ANI     X5  ; RESET   PB6
      AND     SM401  ; Always OFF
      OUT     T5 K10  ; 1-CYCLE OVERTIME
1304  LD      M131  ; 1-CYCLE COMP.PLS
      MOV     T5 D0
1307  LD      M131  ; 1-CYCLE COMP.PLS
      OR      M132  ; OVERRUN DETECT
      ANI     M905  ; GP      Screen-5
      ANI     M904  ; GP      Screen-4
      ANI     M113  ; RKB     1-CYCLE
      ANI     M107  ; INCHING
      ANI     X5  ; RESET   PB6
      OUT     M132  ; OVERRUN DETECT
      OUT     T6 K10  ; OVERRUN DETECT
1319  LD      M213  ; ROBOT   Home
      OR      M9  ; Manual  pulse
      PLS     M131  ; 1-CYCLE COMP.PLS
1323  LD      T6  ; OVERRUN DETECT
      ANI     M214  ; ROBOT   Working Pos
      OR      M133  ; OVER RUN
      ANI     X5  ; RESET   PB6
      ANI     X0  ; MANUAL  PB5
      OUT     M133  ; OVER RUN
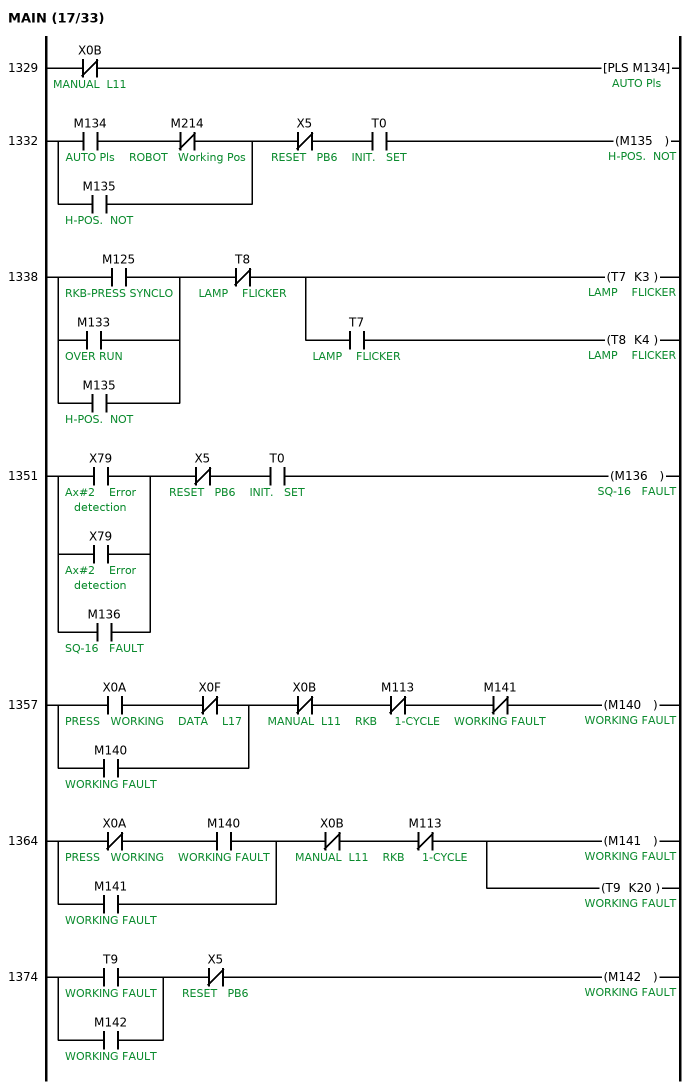
1329  LDI     X0B  ; MANUAL  L11
      PLS     M134  ; AUTO Pls
1332  LD      M134  ; AUTO Pls
      ANI     M214  ; ROBOT   Working Pos
      OR      M135  ; H-POS.  NOT
      ANI     X5  ; RESET   PB6
      AND     T0  ; INIT.   SET
      OUT     M135  ; H-POS.  NOT
1338  LD      M125  ; RKB-PRESS SYNCLO
      OR      M133  ; OVER RUN
      OR      M135  ; H-POS.  NOT
      ANI     T8  ; LAMP    FLICKER
      OUT     T7 K3  ; LAMP    FLICKER
      AND     T7  ; LAMP    FLICKER
      OUT     T8 K4  ; LAMP    FLICKER
1351  LD      X79  ; Ax#2    Error   detection
      OR      X79  ; Ax#2    Error   detection
      OR      M136  ; SQ-16   FAULT
      ANI     X5  ; RESET   PB6
      AND     T0  ; INIT.   SET
      OUT     M136  ; SQ-16   FAULT
1357  LD      X0A  ; PRESS   WORKING
      ANI     X0F  ; DATA    L17
      OR      M140  ; WORKING FAULT
      ANI     X0B  ; MANUAL  L11
      ANI     M113  ; RKB     1-CYCLE
      ANI     M141  ; WORKING FAULT
      OUT     M140  ; WORKING FAULT
1364  LDI     X0A  ; PRESS   WORKING
      AND     M140  ; WORKING FAULT
      OR      M141  ; WORKING FAULT
      ANI     X0B  ; MANUAL  L11
      ANI     M113  ; RKB     1-CYCLE
      OUT     M141  ; WORKING FAULT
      OUT     T9 K20  ; WORKING FAULT
1374  LD      T9  ; WORKING FAULT
      OR      M142  ; WORKING FAULT
      ANI     X5  ; RESET   PB6
      OUT     M142  ; WORKING FAULT
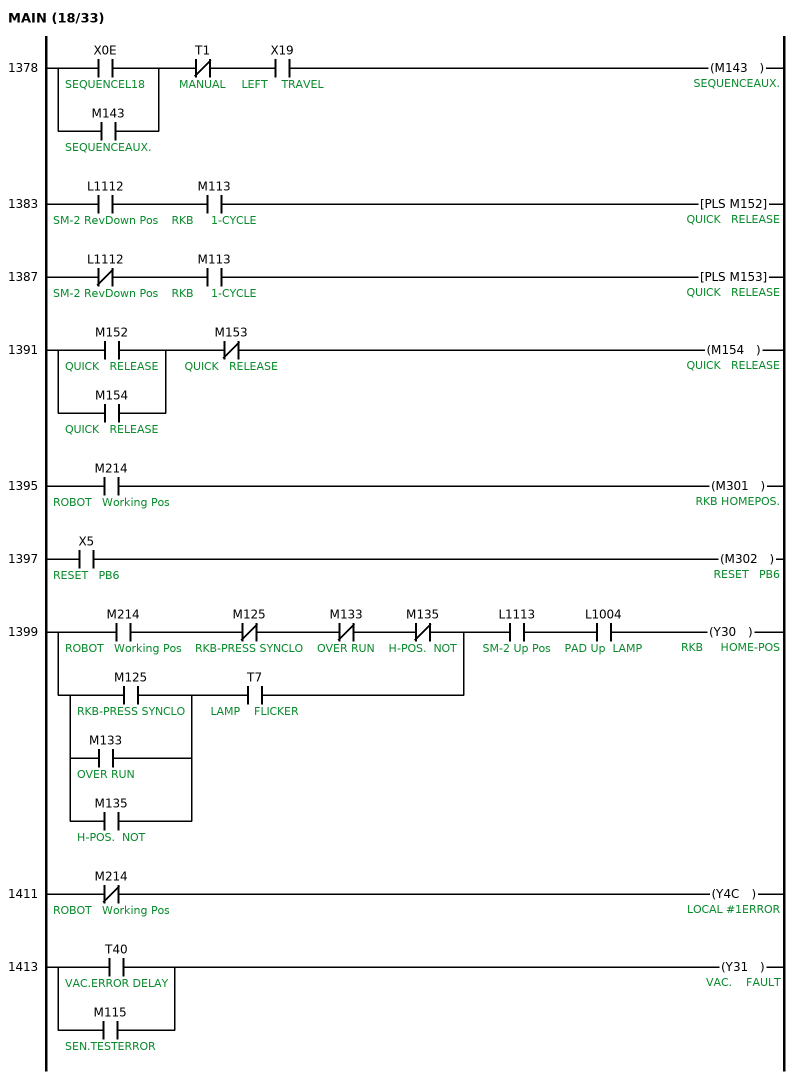
1378  LD      X0E  ; SEQUENCEL18
      OR      M143  ; SEQUENCEAUX.
      ANI     T1  ; MANUAL
      AND     X19  ; LEFT    TRAVEL
      OUT     M143  ; SEQUENCEAUX.
1383  LD      L1112  ; SM-2 RevDown Pos
      AND     M113  ; RKB     1-CYCLE
      PLS     M152  ; QUICK   RELEASE
1387  LDI     L1112  ; SM-2 RevDown Pos
      AND     M113  ; RKB     1-CYCLE
      PLS     M153  ; QUICK   RELEASE
1391  LD      M152  ; QUICK   RELEASE
      OR      M154  ; QUICK   RELEASE
      ANI     M153  ; QUICK   RELEASE
      OUT     M154  ; QUICK   RELEASE
1395  LD      M214  ; ROBOT   Working Pos
      OUT     M301  ; RKB HOMEPOS.
1397  LD      X5  ; RESET   PB6
      OUT     M302  ; RESET   PB6
1399  LD      M214  ; ROBOT   Working Pos
      ANI     M125  ; RKB-PRESS SYNCLO
      ANI     M133  ; OVER RUN
      ANI     M135  ; H-POS.  NOT
      LD      M125  ; RKB-PRESS SYNCLO
      OR      M133  ; OVER RUN
      OR      M135  ; H-POS.  NOT
      AND     T7  ; LAMP    FLICKER
      ORB
      AND     L1113  ; SM-2 Up Pos
      AND     L1004  ; PAD Up  LAMP
      OUT     Y30  ; RKB     HOME-POS
1411  LDI     M214  ; ROBOT   Working Pos
      OUT     Y4C  ; LOCAL #1ERROR
1413  LD      T40  ; VAC.ERROR DELAY
      OR      M115  ; SEN.TESTERROR
      OUT     Y31  ; VAC.    FAULT
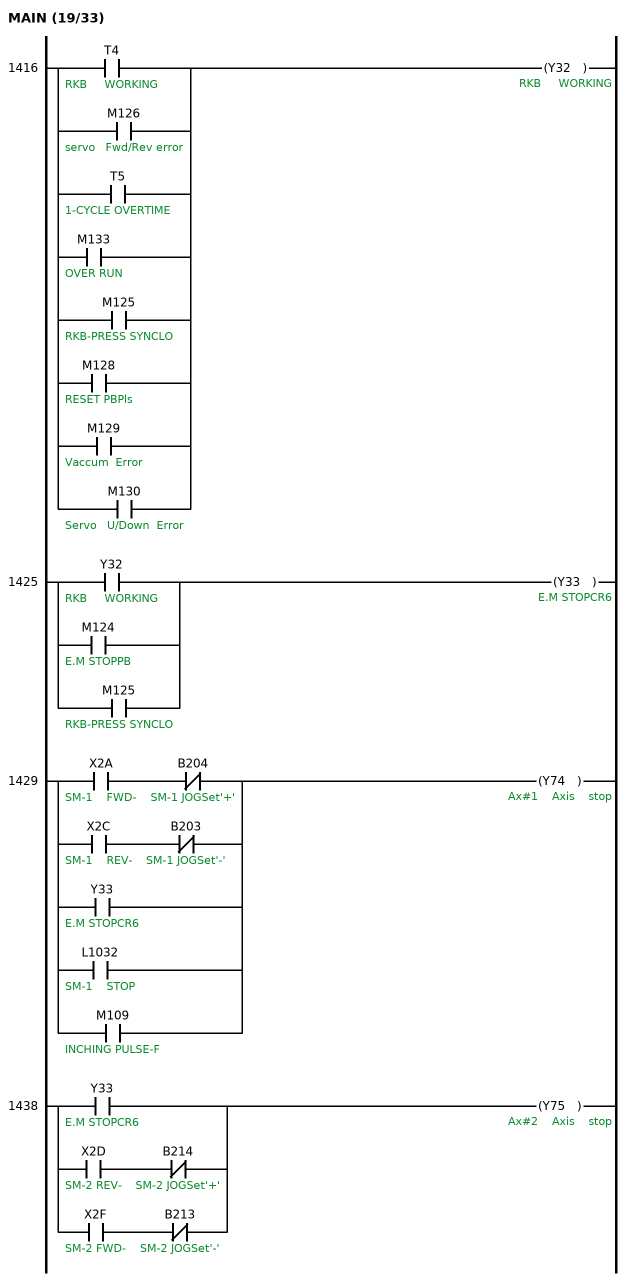
1416  LD      T4  ; RKB     WORKING
      OR      M126  ; servo   Fwd/Rev error
      OR      T5  ; 1-CYCLE OVERTIME
      OR      M133  ; OVER RUN
      OR      M125  ; RKB-PRESS SYNCLO
      OR      M128  ; RESET PBPls
      OR      M129  ; Vaccum  Error
      OR      M130  ; Servo   U/Down  Error
      OUT     Y32  ; RKB     WORKING
1425  LD      Y32  ; RKB     WORKING
      OR      M124  ; E.M STOPPB
      OR      M125  ; RKB-PRESS SYNCLO
      OUT     Y33  ; E.M STOPCR6
1429  LD      X2A  ; SM-1    FWD-
      ANI     B204  ; SM-1 JOGSet'+'
      LD      X2C  ; SM-1    REV-
      ANI     B203  ; SM-1 JOGSet'-'
      ORB
      OR      Y33  ; E.M STOPCR6
      OR      L1032  ; SM-1    STOP
      OR      M109  ; INCHING PULSE-F
      OUT     Y74  ; Ax#1    Axis    stop
1438  LD      Y33  ; E.M STOPCR6
      LD      X2D  ; SM-2 REV-
      ANI     B214  ; SM-2 JOGSet'+'
      ORB
      LD      X2F  ; SM-2 FWD-
      ANI     B213  ; SM-2 JOGSet'-'
      ORB
      OUT     Y75  ; Ax#2    Axis    stop
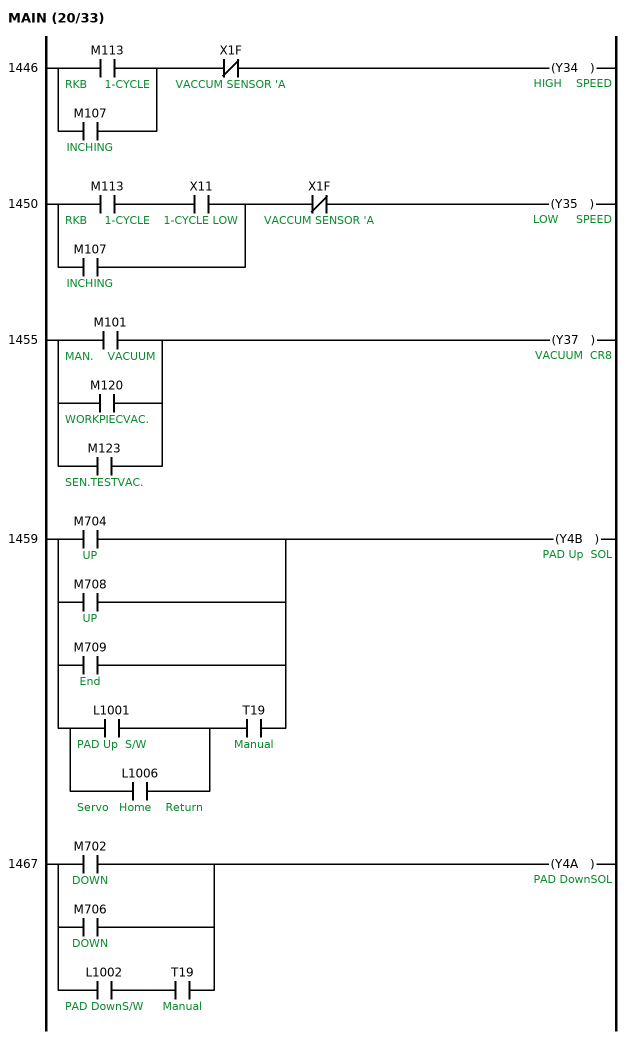
1446  LD      M113  ; RKB     1-CYCLE
      OR      M107  ; INCHING
      ANI     X1F  ; VACCUM SENSOR 'A
      OUT     Y34  ; HIGH    SPEED
1450  LD      M113  ; RKB     1-CYCLE
      AND     X11  ; 1-CYCLE LOW
      OR      M107  ; INCHING
      ANI     X1F  ; VACCUM SENSOR 'A
      OUT     Y35  ; LOW     SPEED
1455  LD      M101  ; MAN.    VACUUM
      OR      M120  ; WORKPIECVAC.
      OR      M123  ; SEN.TESTVAC.
      OUT     Y37  ; VACUUM  CR8
1459  LD      M704  ; UP
      OR      M708  ; UP
      OR      M709  ; End
      LD      L1001  ; PAD Up  S/W
      OR      L1006  ; Servo   Home    Return
      AND     T19  ; Manual
      ORB
      OUT     Y4B  ; PAD Up  SOL
1467  LD      M702  ; DOWN
      OR      M706  ; DOWN
      LD      L1002  ; PAD DownS/W
      AND     T19  ; Manual
      ORB
      OUT     Y4A  ; PAD DownSOL
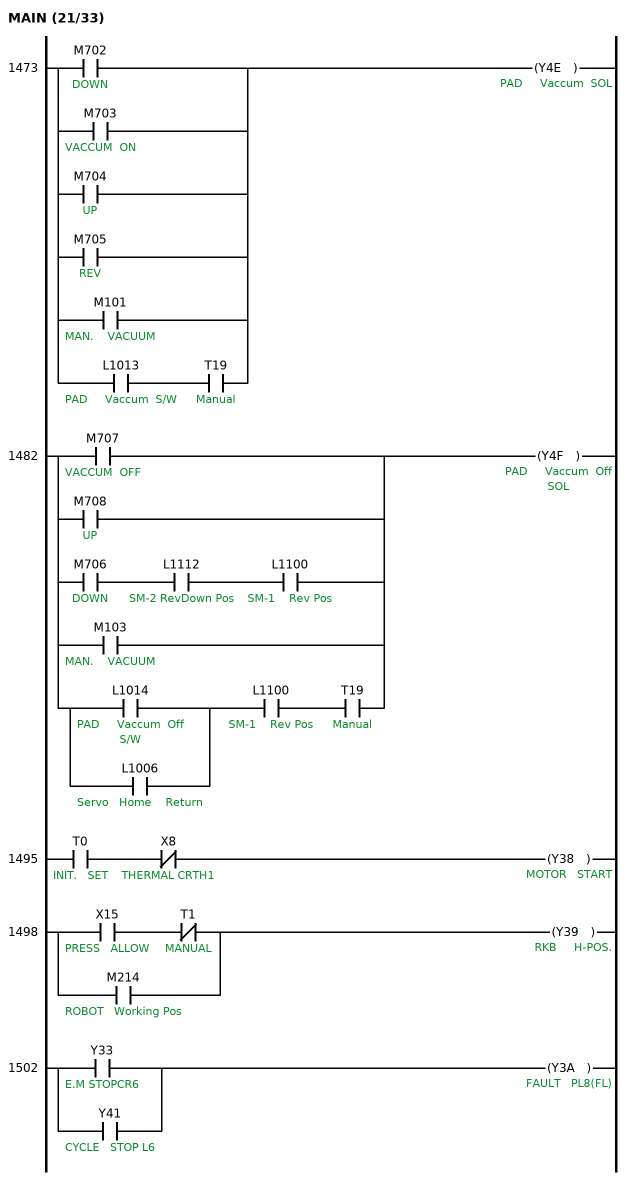
1473  LD      M702  ; DOWN
      OR      M703  ; VACCUM  ON
      OR      M704  ; UP
      OR      M705  ; REV
      OR      M101  ; MAN.    VACUUM
      LD      L1013  ; PAD     Vaccum  S/W
      AND     T19  ; Manual
      ORB
      OUT     Y4E  ; PAD     Vaccum  SOL
1482  LD      M707  ; VACCUM  OFF
      OR      M708  ; UP
      LD      M706  ; DOWN
      AND     L1112  ; SM-2 RevDown Pos
      AND     L1100  ; SM-1    Rev Pos
      ORB
      OR      M103  ; MAN.    VACUUM
      LD      L1014  ; PAD     Vaccum  Off S/W
      OR      L1006  ; Servo   Home    Return
      AND     L1100  ; SM-1    Rev Pos
      AND     T19  ; Manual
      ORB
      OUT     Y4F  ; PAD     Vaccum  Off SOL
1495  LD      T0  ; INIT.   SET
      ANI     X8  ; THERMAL CRTH1
      OUT     Y38  ; MOTOR   START
1498  LD      X15  ; PRESS   ALLOW
      ANI     T1  ; MANUAL
      OR      M214  ; ROBOT   Working Pos
      OUT     Y39  ; RKB     H-POS.
1502  LD      Y33  ; E.M STOPCR6
      OR      Y41  ; CYCLE   STOP L6
      OUT     Y3A  ; FAULT   PL8(FL)
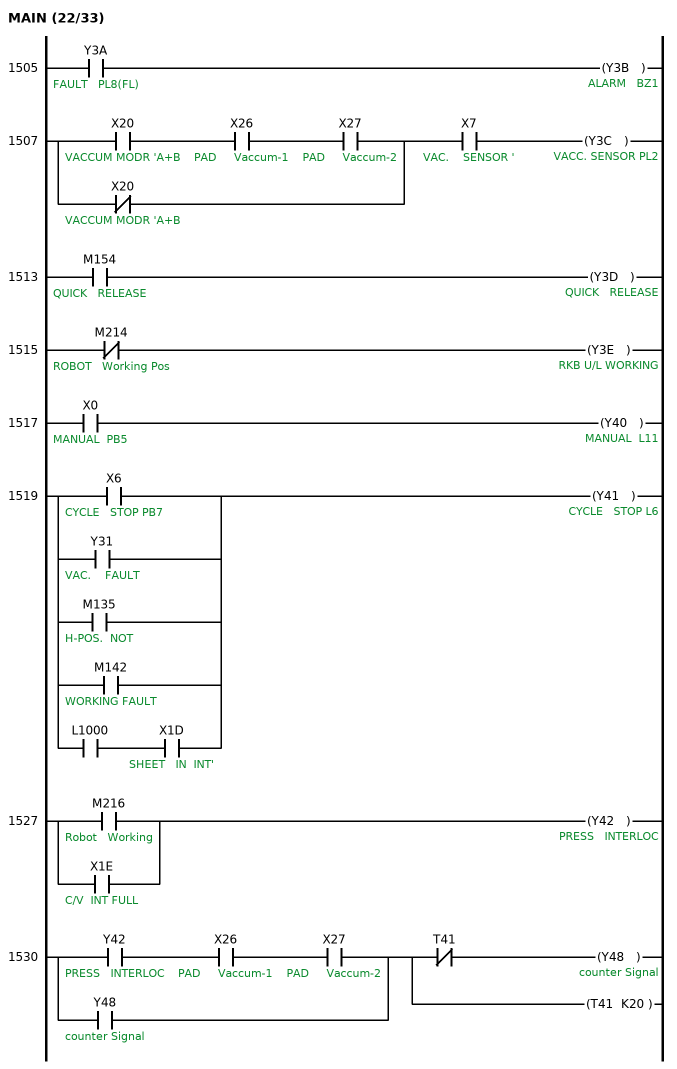
1505  LD      Y3A  ; FAULT   PL8(FL)
      OUT     Y3B  ; ALARM   BZ1
1507  LD      X20  ; VACCUM MODR 'A+B
      AND     X26  ; PAD     Vaccum-1
      AND     X27  ; PAD     Vaccum-2
      ORI     X20  ; VACCUM MODR 'A+B
      AND     X7  ; VAC.    SENSOR '
      OUT     Y3C  ; VACC. SENSOR PL2
1513  LD      M154  ; QUICK   RELEASE
      OUT     Y3D  ; QUICK   RELEASE
1515  LDI     M214  ; ROBOT   Working Pos
      OUT     Y3E  ; RKB U/L WORKING
1517  LD      X0  ; MANUAL  PB5
      OUT     Y40  ; MANUAL  L11
1519  LD      X6  ; CYCLE   STOP PB7
      OR      Y31  ; VAC.    FAULT
      OR      M135  ; H-POS.  NOT
      OR      M142  ; WORKING FAULT
      LD      L1000
      AND     X1D  ; SHEET   IN  INT'
      ORB
      OUT     Y41  ; CYCLE   STOP L6
1527  LD      M216  ; Robot   Working
      OR      X1E  ; C/V  INT FULL
      OUT     Y42  ; PRESS   INTERLOC
1530  LD      Y42  ; PRESS   INTERLOC
      AND     X26  ; PAD     Vaccum-1
      AND     X27  ; PAD     Vaccum-2
      OR      Y48  ; counter Signal
      MPS
      ANI     T41
      OUT     Y48  ; counter Signal
      MPP
      OUT     T41 K20
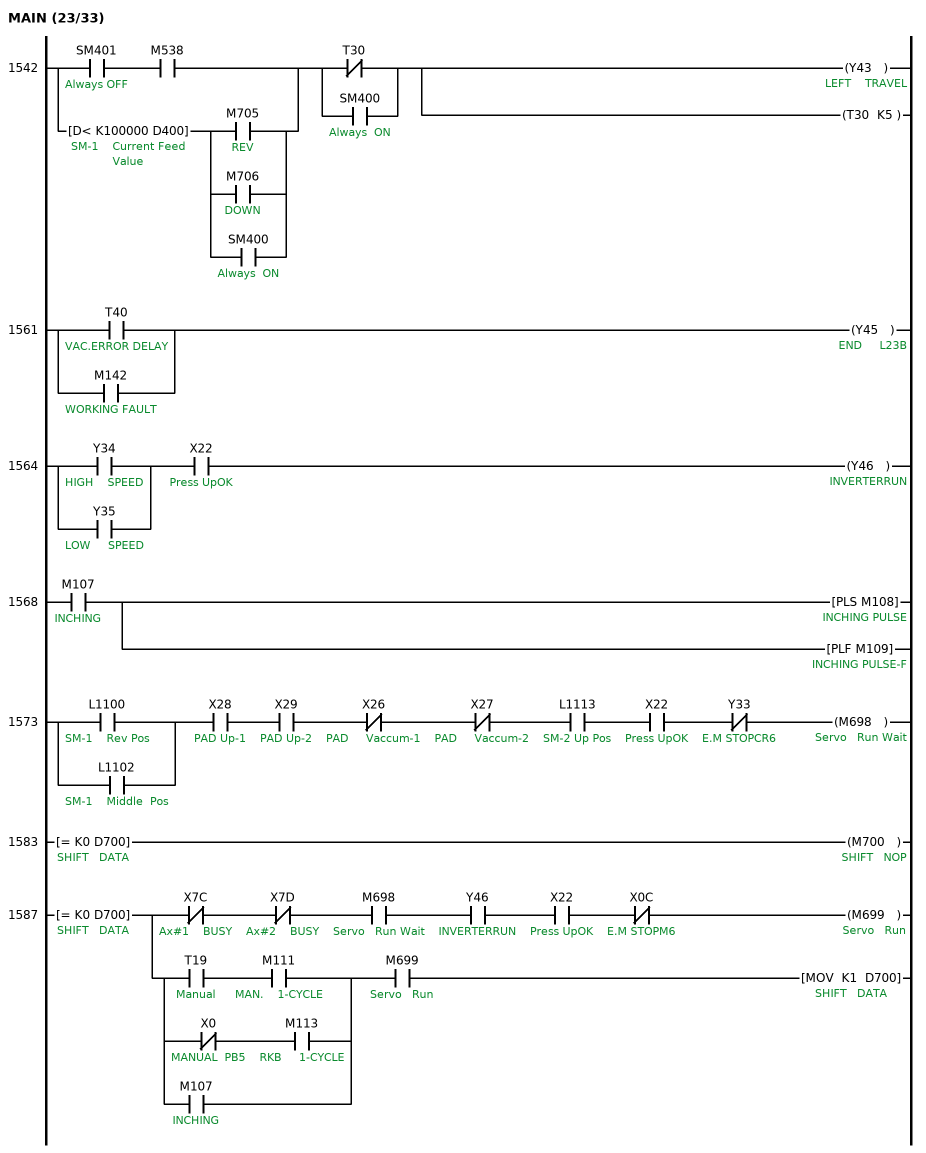
1542  LD      SM401  ; Always OFF
      AND     M538
      LDD<    K100000 D400  ; SM-1    Current Feed    Value
      LD      M705  ; REV
      OR      M706  ; DOWN
      OR      SM400  ; Always  ON
      ANB
      ORB
      LDI     T30
      OR      SM400  ; Always  ON
      ANB
      OUT     Y43  ; LEFT    TRAVEL
      OUT     T30 K5
1561  LD      T40  ; VAC.ERROR DELAY
      OR      M142  ; WORKING FAULT
      OUT     Y45  ; END     L23B
1564  LD      Y34  ; HIGH    SPEED
      OR      Y35  ; LOW     SPEED
      AND     X22  ; Press UpOK
      OUT     Y46  ; INVERTERRUN
1568  LD      M107  ; INCHING
      PLS     M108  ; INCHING PULSE
      PLF     M109  ; INCHING PULSE-F
1573  LD      L1100  ; SM-1    Rev Pos
      OR      L1102  ; SM-1    Middle  Pos
      AND     X28  ; PAD Up-1
      AND     X29  ; PAD Up-2
      ANI     X26  ; PAD     Vaccum-1
      ANI     X27  ; PAD     Vaccum-2
      AND     L1113  ; SM-2 Up Pos
      AND     X22  ; Press UpOK
      ANI     Y33  ; E.M STOPCR6
      OUT     M698  ; Servo   Run Wait
1583  LD=     K0 D700  ; SHIFT   DATA
      OUT     M700  ; SHIFT   NOP
1587  LD=     K0 D700  ; SHIFT   DATA
      MPS
      ANI     X7C  ; Ax#1    BUSY
      ANI     X7D  ; Ax#2    BUSY
      AND     M698  ; Servo   Run Wait
      AND     Y46  ; INVERTERRUN
      AND     X22  ; Press UpOK
      ANI     X0C  ; E.M STOPM6
      OUT     M699  ; Servo   Run
      MPP
      LD      T19  ; Manual
      AND     M111  ; MAN.    1-CYCLE
      LDI     X0  ; MANUAL  PB5
      AND     M113  ; RKB     1-CYCLE
      ORB
      OR      M107  ; INCHING
      ANB
      AND     M699  ; Servo   Run
      MOV     K1 D700
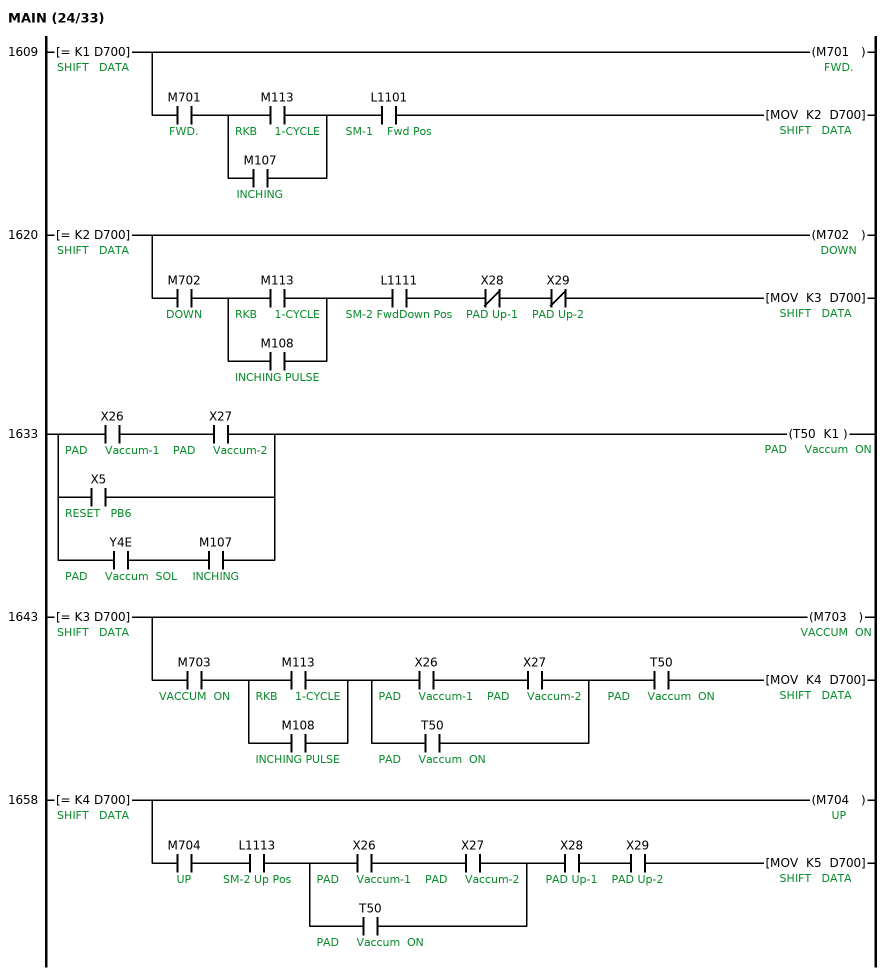
1609  LD=     K1 D700  ; SHIFT   DATA
      OUT     M701  ; FWD.
      AND     M701  ; FWD.
      LD      M113  ; RKB     1-CYCLE
      OR      M107  ; INCHING
      ANB
      AND     L1101  ; SM-1    Fwd Pos
      MOV     K2 D700
1620  LD=     K2 D700  ; SHIFT   DATA
      OUT     M702  ; DOWN
      AND     M702  ; DOWN
      LD      M113  ; RKB     1-CYCLE
      OR      M108  ; INCHING PULSE
      ANB
      AND     L1111  ; SM-2 FwdDown Pos
      ANI     X28  ; PAD Up-1
      ANI     X29  ; PAD Up-2
      MOV     K3 D700
1633  LD      X26  ; PAD     Vaccum-1
      AND     X27  ; PAD     Vaccum-2
      OR      X5  ; RESET   PB6
      LD      Y4E  ; PAD     Vaccum  SOL
      AND     M107  ; INCHING
      ORB
      OUT     T50 K1  ; PAD     Vaccum  ON
1643  LD=     K3 D700  ; SHIFT   DATA
      OUT     M703  ; VACCUM  ON
      AND     M703  ; VACCUM  ON
      LD      M113  ; RKB     1-CYCLE
      OR      M108  ; INCHING PULSE
      ANB
      LD      X26  ; PAD     Vaccum-1
      AND     X27  ; PAD     Vaccum-2
      OR      T50  ; PAD     Vaccum  ON
      ANB
      AND     T50  ; PAD     Vaccum  ON
      MOV     K4 D700
1658  LD=     K4 D700  ; SHIFT   DATA
      OUT     M704  ; UP
      AND     M704  ; UP
      AND     L1113  ; SM-2 Up Pos
      LD      X26  ; PAD     Vaccum-1
      AND     X27  ; PAD     Vaccum-2
      OR      T50  ; PAD     Vaccum  ON
      ANB
      AND     X28  ; PAD Up-1
      AND     X29  ; PAD Up-2
      MOV     K5 D700
